(* CODESYS project HeatSeal.xml

Project tree, tasks and I/O mapping:
  function block HeatSeal [CFC]
*)

// HeatSeal
FUNCTION_BLOCK HeatSeal
//  .					.					.
VAR_INPUT
	Enable: 			BOOL;
	Open: 				BOOL;
	Close: 				BOOL;
	OpenSensor: 		BOOL;
	CloseSensor: 		BOOL;
	Stop: 				BOOL;
	Reset: 				BOOL;
END_VAR
VAR_OUTPUT
	Forward: 			BOOL;
	Reverse: 			BOOL;
	Brake: 				BOOL;
	Closed: 			BOOL;
	Opened: 			BOOL;
END_VAR
VAR
	_Sequence: 			HeatSealSequence;
	_ManualOpen: 		BOOL;
	_ManualClose: 		BOOL;
	_ManualStop: 		BOOL;
	_ManualReset: 		BOOL;
	_EnableOpen: 		BOOL;
	_EnableClose: 		BOOL;
END_VAR
VAR // added by the converter: edge detectors and wires of the graphical bodies
    _w1 : BOOL;
    _w2, _w3 : ANY;
END_VAR

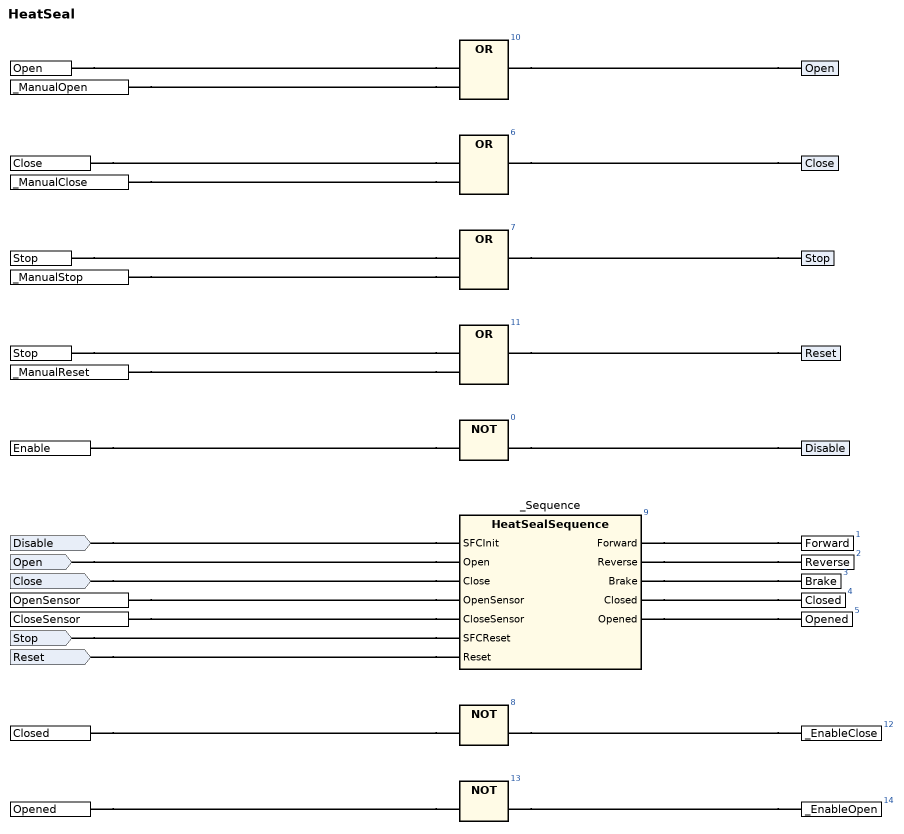
// note: 18 stored wires end on pins the file does not list and are not shown
Forward := _Sequence.Forward;
Reverse := _Sequence.Reverse;
Brake := _Sequence.Brake;
Closed := _Sequence.Closed;
Opened := _Sequence.Opened;
_w1 := NOT Closed;
_Sequence(
    SFCInit := NOT Enable,
    Open := _w2,
    Close := Close OR _ManualClose,
    OpenSensor := OpenSensor,
    CloseSensor := CloseSensor,
    SFCReset := Stop OR _ManualStop,
    Reset := _w3); // HeatSealSequence
_w2 := Open OR _ManualOpen;
_w3 := Stop OR _ManualReset;
_EnableClose := _w1;
_EnableOpen := NOT Opened;

END_FUNCTION_BLOCK
